(* CoDeSys 2.3.9.37 project: Cap6_9.pro *)
(* Libraries: Standard.LIB 4.10.05 12:14:46 *)

(* Global variable list: Global_Variables *)
VAR_GLOBAL
     (* Entradas *)
	A: BOOL;
	B: BOOL;

      (* Salidas *)
	salrojo: BOOL;
       salverde:BOOL;

END_VAR

(* POU PLC_PRG, FBD *)
PROGRAM PLC_PRG
VAR

END_VAR
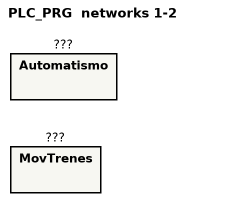
_FBD_ (* Function Block Diagram *)
NETWORK 1
	???:Automatismo()
NETWORK 2
	???:MovTrenes()
_END_FBD_
END_PROGRAM

(* POU Automatismo, LD *)
PROGRAM Automatismo
VAR

END_VAR
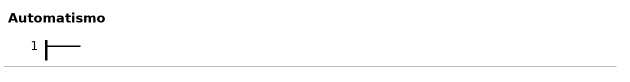
_LD_ (* Ladder Diagram *)
NETWORK 1
	*
_END_LD_
(* the same logic as Structured Text *)
(* Network 1 *)
END_PROGRAM

(* POU MovTrenes, ST *)
PROGRAM MovTrenes
VAR
  ENTRA_IZQ:BOOL;
	tren_izq: BOOL;
	posx: INT :=-550;
	ENTRA_DER: BOOL;
	tren_der: BOOL;
END_VAR
IF (ENTRA_IZQ=TRUE) AND (tren_der=FALSE) THEN
    tren_izq:=TRUE;
ELSE
   IF  (ENTRA_DER=TRUE) AND (tren_izq=FALSE) AND (tren_der=FALSE) THEN
       tren_der:=TRUE;
      posx:=390;
   END_IF
END_IF

IF (tren_izq=TRUE) THEN
   posx:=posx+2;
END_IF


IF (tren_der=TRUE) THEN
   posx:=posx-2;
END_IF

IF (posx>-430) AND (posx<-100) THEN
   A:=TRUE;
ELSE
   A:=FALSE;
END_IF

IF (posx>16) AND (posx<350) THEN
   B:=TRUE;
ELSE
   B:=FALSE;
END_IF

IF (posx=400) AND (tren_izq=TRUE)  THEN
    tren_izq:=FALSE;
    posx:=-550;
END_IF


IF (posx=-500) AND (tren_der=TRUE) THEN
    tren_der:=FALSE;
    posx:=-550;
END_IF
END_PROGRAM

(* Visualisation Tren
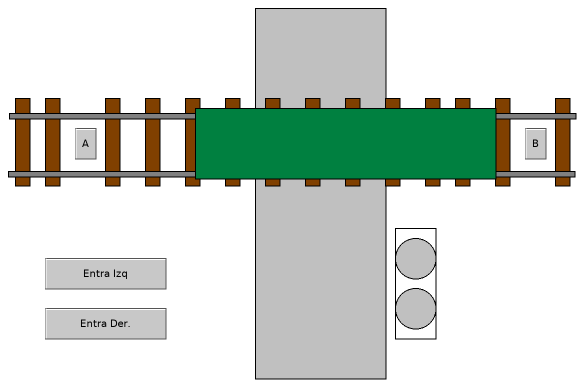
button at (60,120)-(81,151): text "A"; toggles PLC_PRG.A
button at (510,120)-(531,151): text "B"; toggles PLC_PRG.B
ellipse at (380,230)-(421,271): alarm colour if salrojo
ellipse at (380,280)-(421,321): alarm colour if salverde
rounded rectangle at (180,100)-(481,171): x offset MovTrenes.posx
button at (30,250)-(151,281): text "Entra Izq"; taps MovTrenes.ENTRA_IZQ
button at (30,300)-(151,331): text "Entra Der."; taps MovTrenes.ENTRA_DER
18 more shapes without text or variables
*)
